{attribute addProperty BoxType "AX8620-1000-0027"}
{attribute addProperty Id "StatuswordAT %I*Statusword_177FE35F162"}
{attribute addProperty CRC "3243559737"}
{attribute addProperty SizeInBites "16"}
{attribute addProperty SizeInBytes "2"}
TYPE PSM_PSM_Statusword_C154CB39 :
STRUCT
	{attribute addProperty Name "Statusword"}
	Statusword AT %I* : Statusword_177FE35F;
END_STRUCT
END_TYPE

(* stored: Version 1.2.0.0, ProductVersion 3.1.4024.9
   DUT PSM_PSM_Statusword_C154CB39: Id {7e8dd210-e87c-4205-b6c8-92394e83af14} *)
